FUNCTION_BLOCK FB_TestRange EXTENDS TcUnit.FB_TestSuite

testRange100to1000_min();
testRange100to1000_max();
testRange100to1000_mid();
testRange100to1000_OverMax();
testRange100to1000_UnderMin();

// Bounds
testCheckBounds_valid();
testCheckBounds_invalid();

METHOD testCheckBounds_invalid
VAR
	
	Actual  	: BOOL; 
	Expected 	: BOOL;
	
	arrayIn		: ARRAY[0..5] OF INT;
END_VAR
TEST('testCheckBounds_invalid');

// Act
Actual := F_IN_BOUNDS_ARRAY_INT(6, arrayIn); 

// Arrange
Expected := FALSE;

// Assert
AssertEquals_BOOL( Expected := Expected, 
				  Actual := Actual,
			 	  Message := 'testCheckBounds_invalid Failed to get in bounds');		 
			 
			 
TEST_FINISHED();
END_METHOD

METHOD testCheckBounds_valid
VAR
	
	Actual  	: BOOL; 
	Expected 	: BOOL;
	
	arrayIn		: ARRAY[0..5] OF INT;
END_VAR
TEST('testCheckBounds_valid');

// Act
Actual := F_IN_BOUNDS_ARRAY_INT(5, arrayIn); 

// Arrange
Expected := TRUE;

// Assert
AssertEquals_BOOL( Expected := Expected, 
				  Actual := Actual,
			 	  Message := 'testCheckBounds_valid Failed to get in bounds');		 
			 
			 
TEST_FINISHED();
END_METHOD

METHOD testRange100to1000_max
VAR
	iValue		: INT := 100;
	
	iValue_Max	: INT := 100;
	iValue_min	: INT := 0;
	
	iRange_max	: INT := 1000;
	iRange_min	: INT := 100;
	
	Actual		: INT;
	Expected  	: INT;
	
	ActualVarInfo : __SYSTEM.VAR_INFO;
END_VAR
TEST('testRange100to1000_max');

// Act
Actual := F_GET_IN_RANGE_INT(iValue, iRange_Max, iRange_Min, iValue_Max, iValue_Min); 

// Arrange
Expected := 1000;

// Assert
AssertEquals_INT( Expected := Expected, 
				  Actual := Actual,
			 	  Message := 'testRange100to1000_max Failed to get in range INT');

ActualVarInfo :=__VARINFO(Actual);
 
AssertTrue(  Condition := ActualVarInfo.TypeName = 'INT',
			  Message := 'testRange100to1000_max Failed in type INT');
			 
			 
			 
TEST_FINISHED();
END_METHOD

METHOD testRange100to1000_mid
VAR
	iValue		: INT := 50;
	
	iValue_Max	: INT := 100;
	iValue_min	: INT := 0;
	
	iRange_max	: INT := 1000;
	iRange_min	: INT := 100;
	
	Actual		: INT;
	Expected  	: INT;
END_VAR
TEST('testRange100to1000_mid');

// Act
Actual := F_GET_IN_RANGE_INT(iValue, iRange_Max, iRange_Min, iValue_Max, iValue_Min); 

// Arrange
Expected := 550;

// Assert
AssertEquals_INT( Expected := Expected, 
				  Actual := Actual,
			 	  Message := 'testRange100to1000_mid Failed to get in range INT');
			 
			 
			 
TEST_FINISHED();
END_METHOD

METHOD testRange100to1000_min
VAR
	iValue		: INT := 0;
	
	iValue_Max	: INT := 100;
	iValue_min	: INT := 0;
	
	iRange_max	: INT := 1000;
	iRange_min	: INT := 100;
	
	Actual		: INT;
	Expected  	: INT;
END_VAR
TEST('testRange100to1000_min');

// Act
Actual := F_GET_IN_RANGE_INT(iValue, iRange_Max, iRange_Min, iValue_Max, iValue_Min); 

// Arrange
Expected := 100;

// Assert
AssertEquals_INT( Expected := Expected, 
				  Actual := Actual,
			 	  Message := 'testRange100to1000_min Failed to get in range INT');
			 
			 
			 
TEST_FINISHED();
END_METHOD

METHOD testRange100to1000_OverMax
VAR
	iValue		: INT := 200;
	
	iValue_Max	: INT := 100;
	iValue_min	: INT := 0;
	
	iRange_max	: INT := 1000;
	iRange_min	: INT := 100;
	
	Actual		: INT;
	Expected  	: INT;
	
	ActualVarInfo : __SYSTEM.VAR_INFO;
END_VAR
TEST('testRange100to1000_OverMax');

// Act
Actual := F_GET_IN_RANGE_INT(iValue, iRange_Max, iRange_Min, iValue_Max, iValue_Min); 

// Arrange
Expected := iRange_max;

// Assert
AssertEquals_INT( Expected := Expected, 
				  Actual := Actual,
			 	  Message := 'testRange100to1000_OverMax Failed to get in range INT');			 
			 
TEST_FINISHED();
END_METHOD

METHOD testRange100to1000_UnderMin
VAR
	iValue		: INT := -100;
	
	iValue_Max	: INT := 100;
	iValue_min	: INT := 0;
	
	iRange_max	: INT := 1000;
	iRange_min	: INT := 100;
	
	Actual		: INT;
	Expected  	: INT;
	
	ActualVarInfo : __SYSTEM.VAR_INFO;
END_VAR
TEST('testRange100to1000_UnderMin');

// Act
Actual := F_GET_IN_RANGE_INT(iValue, iRange_Max, iRange_Min, iValue_Max, iValue_Min); 

// Arrange
Expected := iRange_min;

// Assert
AssertEquals_INT( Expected := Expected, 
				  Actual := Actual,
			 	  Message := 'testRange100to1000_UnderMin Failed to get in range INT');			 
			 
TEST_FINISHED();
END_METHOD

END_FUNCTION_BLOCK

(* stored: Version 1.1.0.1, ProductVersion 3.1.4024.9
   POU FB_TestRange: Id {905c3600-7cc8-425a-9a8d-1f2dcb1a9cd4}, SpecialFunc None
   Method testCheckBounds_invalid: Id {4e52e6ee-a9bd-44d5-b575-0f3c3d47632a}
   Method testCheckBounds_valid: Id {7e8a22f1-ff1c-4dd7-9eec-e3599d699a46}
   Method testRange100to1000_max: Id {e3272f19-c110-4b42-88ab-a38ea1065e51}
   Method testRange100to1000_mid: Id {5b5fc52d-dfcc-4767-a063-8bbcc5a8a407}
   Method testRange100to1000_min: Id {c94efede-8e05-4cac-91ad-0f8f71b78b03}
   Method testRange100to1000_OverMax: Id {316ffd6d-1509-4599-b2f2-44d2c76dbe5b}
   Method testRange100to1000_UnderMin: Id {08d8553f-0e41-4d95-b548-1755c0fad12f} *)
